FUNCTION_BLOCK _ETcVnBarcodeSearchDirection_TestSuite EXTENDS TcUnit.FB_TestSuite
VAR
END_VAR

TestAddress();
TestClearReference();
TestClone();
TestTypeNameReturnsExpected();
TestIdentifierReturnsExpected();
TestMakeReferenceToFollowsReference();
TestMakeReferenceToUpdatesReference();
TestSize();
TestValueReturnsExpectedAfterInit();
TestValueReturnsExpectedAfterChange();
TestSerializeTypeWith();
TestSerializeWith();
TestTryDeserializeFrom();
TestTryMakeReferenceToFollowsReference();
TestTryMakeReferenceToUpdatesReference();

METHOD PUBLIC TestAddress
VAR
    _type : _ETcVnBarcodeSearchDirection(ETcVnBarcodeSearchDirection.TCVN_BSD_ANY);
    notExpected : PVOID := 0;
    actual : PVOID;
END_VAR
TEST('TestAddress');

actual := _type.Address;

AssertFalse(
    Condition := (notExpected = actual),
    Message := 'Type did not return a valid address.'
);

TEST_FINISHED();
END_METHOD

METHOD PUBLIC TestClearReference
VAR
    _type : _ETcVnBarcodeSearchDirection(ETcVnBarcodeSearchDirection.TCVN_BSD_ANY);
	target : ETcVnBarcodeSearchDirection := ETcVnBarcodeSearchDirection.TCVN_BSD_ANY;
    expected : ETcVnBarcodeSearchDirection := ETcVnBarcodeSearchDirection.TCVN_BSD_ANY;
    actual : ETcVnBarcodeSearchDirection;
END_VAR
TEST('TestClearReference');

_type.MakeReferenceTo(target);
_type.ClearReference();
target := ETcVnBarcodeSearchDirection.TCVN_BSD_HORIZONTAL;

actual := _type.Value;

AssertEquals(
    Expected := expected,
    Actual := actual,
    Message := 'Value continued to follow target.'
);

TEST_FINISHED();
END_METHOD

METHOD PUBLIC TestClone
VAR
    _type : _ETcVnBarcodeSearchDirection(ETcVnBarcodeSearchDirection.TCVN_BSD_ANY);
	clone : I_Datatype;
	isValidClone : BOOL;
	compareResult : DINT;
END_VAR
TEST('TestClone');

clone := _type.Clone();

isValidClone := clone <> 0;

IF isValidClone THEN
	compareResult := memcmp(_type.Address, clone.Address, clone.Size);
END_IF

AssertTrue(
	Condition := isValidClone,
	Message := 'Clone did not produce a clone'
);

AssertEquals_DINT(
	Expected := 0,
    Actual := compareResult,
    Message := 'Clone did not return a valid clone.'
);

clone.Dispose();

TEST_FINISHED();
END_METHOD

METHOD PUBLIC TestIdentifierReturnsExpected
VAR
    _type : _ETcVnBarcodeSearchDirection(ETcVnBarcodeSearchDirection.TCVN_BSD_ANY);
    expected : STRING := 'ETcVnBarcodeSearchDirection';
    actual : STRING;
END_VAR
TEST('TestIdentifierReturnsExpected');

actual := _type.Identifier;

AssertEquals_STRING(
    Expected := expected,
    Actual := actual,
    Message := 'Type did not return correct iec type.'
);

TEST_FINISHED();
END_METHOD

METHOD PUBLIC TestMakeReferenceToFollowsReference
VAR
    _type : _ETcVnBarcodeSearchDirection(ETcVnBarcodeSearchDirection.TCVN_BSD_ANY);
	target : ETcVnBarcodeSearchDirection := ETcVnBarcodeSearchDirection.TCVN_BSD_ANY;
    expected : ETcVnBarcodeSearchDirection := ETcVnBarcodeSearchDirection.TCVN_BSD_HORIZONTAL;
    actual : ETcVnBarcodeSearchDirection;
END_VAR
TEST('TestMakeReferenceToFollowsReference');

_type.MakeReferenceTo(target);
target := ETcVnBarcodeSearchDirection.TCVN_BSD_HORIZONTAL;

actual := _type.Value;

AssertEquals(
    Expected := expected,
    Actual := actual,
    Message := 'Value did not follow target change.'
);

TEST_FINISHED();
END_METHOD

METHOD PUBLIC TestMakeReferenceToUpdatesReference
VAR
    _type : _ETcVnBarcodeSearchDirection(ETcVnBarcodeSearchDirection.TCVN_BSD_ANY);
	target : ETcVnBarcodeSearchDirection := ETcVnBarcodeSearchDirection.TCVN_BSD_ANY;
    expected : ETcVnBarcodeSearchDirection := ETcVnBarcodeSearchDirection.TCVN_BSD_HORIZONTAL;
    actual : ETcVnBarcodeSearchDirection;
END_VAR
TEST('TestMakeReferenceToUpdatesReference');

_type.MakeReferenceTo(target);
_type.Value := ETcVnBarcodeSearchDirection.TCVN_BSD_HORIZONTAL;

actual := target;

AssertEquals(
    Expected := expected,
    Actual := actual,
    Message := 'Value did not update target.'
);

TEST_FINISHED();
END_METHOD

METHOD PUBLIC TestSerializeTypeWith
VAR
    _type : _ETcVnBarcodeSearchDirection(ETcVnBarcodeSearchDirection.TCVN_BSD_ANY);
    serializer : JsonSerializer;
    expected : STRING(500) := '{"typeName":"ENUM","identifier":"ETcVnBarcodeSearchDirection","enumerations":["TCVN_BSD_ANY","TCVN_BSD_HORIZONTAL","TCVN_BSD_VERTICAL"],"baseType":{"typeName":"UDINT","minValue":0,"maxValue":4294967295,"isSigned":false,"isFloat":false}}'; 
    actual : STRING(500);
END_VAR
TEST('TestSerializeTypeWith');

serializer.Reset();
_type.SerializeTypeWith(serializer);
serializer.TryGetSerializedData(ADR(actual), SIZEOF(actual));

AssertEquals_STRING(
    Expected := expected,
    Actual := actual,
    Message := 'Serialization of type did not return correct string.'
);

TEST_FINISHED();
END_METHOD

METHOD PUBLIC TestSerializeWith
VAR
    _type : _ETcVnBarcodeSearchDirection(ETcVnBarcodeSearchDirection.TCVN_BSD_ANY);
    serializer : JsonSerializer;
    expected : STRING := '"TCVN_BSD_ANY"';
    actual : STRING(500);
END_VAR
TEST('TestSerializeWith');

serializer.Reset();
_type.SerializeWith(serializer);
serializer.TryGetSerializedData(ADR(actual), SIZEOF(actual));

AssertEquals_STRING(
    Expected := expected,
    Actual := actual,
    Message := 'Serialization of type data did not return correct string.'
);

TEST_FINISHED();
END_METHOD

METHOD PUBLIC TestSize
VAR
    _type : _ETcVnBarcodeSearchDirection(ETcVnBarcodeSearchDirection.TCVN_BSD_ANY);
    expected : UDINT := SIZEOF(ETcVnBarcodeSearchDirection);
    actual : UDINT;
END_VAR
TEST('TestSize');

actual := _type.Size;

AssertEquals_UDINT(
    Expected := Expected,
    Actual := actual,
    Message := 'Type did not return the correct size.'
);

TEST_FINISHED();
END_METHOD

METHOD PUBLIC TestTryDeserializeFrom
VAR
    deserializer : JsonDeserializer;
    feedback : DeserializerFeedback;
    json : STRING := '"TCVN_BSD_ANY"';
    _type : _ETcVnBarcodeSearchDirection(ETcVnBarcodeSearchDirection.TCVN_BSD_ANY);
    expected : ETcVnBarcodeSearchDirection := ETcVnBarcodeSearchDirection.TCVN_BSD_ANY;
    actual : ETcVnBarcodeSearchDirection;
 END_VAR
TEST('TestTryDeserializeFrom');

deserializer.Reset();
deserializer.TryLoad(json);
_type.TryDeserializeFrom(Deserializer, Feedback);

actual := _type.Value;

AssertEquals(
    Expected := expected,
    Actual := actual,
    Message := 'Type did not deserialize correctly.'
);

TEST_FINISHED();
END_METHOD

METHOD PUBLIC TestTryMakeReferenceToFollowsReference
VAR
    _type : _ETcVnBarcodeSearchDirection(ETcVnBarcodeSearchDirection.TCVN_BSD_ANY);
	target : _ETcVnBarcodeSearchDirection(ETcVnBarcodeSearchDirection.TCVN_BSD_ANY);
    expected : ETcVnBarcodeSearchDirection := ETcVnBarcodeSearchDirection.TCVN_BSD_HORIZONTAL;
    actual : ETcVnBarcodeSearchDirection;
END_VAR
TEST('TestTryMakeReferenceToFollowsReference');

_type.TryMakeReferenceTo(target);
target.Value := ETcVnBarcodeSearchDirection.TCVN_BSD_HORIZONTAL;

actual := _type.Value;

AssertEquals(
    Expected := expected,
    Actual := actual,
    Message := 'Value did not follow target change.'
);

TEST_FINISHED();
END_METHOD

METHOD PUBLIC TestTryMakeReferenceToUpdatesReference
VAR
    _type : _ETcVnBarcodeSearchDirection(ETcVnBarcodeSearchDirection.TCVN_BSD_ANY);
	target : _ETcVnBarcodeSearchDirection(ETcVnBarcodeSearchDirection.TCVN_BSD_ANY);
    expected : ETcVnBarcodeSearchDirection := ETcVnBarcodeSearchDirection.TCVN_BSD_HORIZONTAL;
    actual : ETcVnBarcodeSearchDirection;
END_VAR
TEST('TestTryMakeReferenceToUpdatesReference');

_type.TryMakeReferenceTo(target);
_type.Value := ETcVnBarcodeSearchDirection.TCVN_BSD_HORIZONTAL;

actual := target.Value;

AssertEquals(
    Expected := expected,
    Actual := actual,
    Message := 'Value did not update target.'
);

TEST_FINISHED();
END_METHOD

METHOD PUBLIC TestTypeNameReturnsExpected
VAR
    _type : _ETcVnBarcodeSearchDirection(ETcVnBarcodeSearchDirection.TCVN_BSD_ANY);
    expected : STRING := 'ENUM';
    actual : STRING;
END_VAR
TEST('TestTypeNameReturnsExpected');

actual := _type.TypeName;

AssertEquals_STRING(
    Expected := expected,
    Actual := actual,
    Message := 'Type did not return correct iec type.'
);

TEST_FINISHED();
END_METHOD

METHOD PUBLIC TestValueReturnsExpectedAfterChange
VAR
    _type : _ETcVnBarcodeSearchDirection(ETcVnBarcodeSearchDirection.TCVN_BSD_ANY);
    expected : ETcVnBarcodeSearchDirection := ETcVnBarcodeSearchDirection.TCVN_BSD_HORIZONTAL;
    actual : ETcVnBarcodeSearchDirection;
END_VAR
TEST('TestValueReturnsExpectedAfterChange');

_type.Value := ETcVnBarcodeSearchDirection.TCVN_BSD_HORIZONTAL;

actual := _type.Value;

AssertEquals(
    Expected := expected,
    Actual := actual,
    Message := 'Expected value not returned after change.'
);

TEST_FINISHED();
END_METHOD

METHOD PUBLIC TestValueReturnsExpectedAfterInit
VAR
    _type : _ETcVnBarcodeSearchDirection(ETcVnBarcodeSearchDirection.TCVN_BSD_ANY);
    expected : ETcVnBarcodeSearchDirection := ETcVnBarcodeSearchDirection.TCVN_BSD_ANY;
    actual : ETcVnBarcodeSearchDirection;
END_VAR
TEST('TestValueReturnsExpectedAfterInit');

actual := _type.Value;

AssertEquals(
    Expected := expected,
    Actual := actual,
    Message := 'Expected value not returned after Init.'
);

TEST_FINISHED();
END_METHOD

END_FUNCTION_BLOCK

(* stored: Version 1.1.0.1, ProductVersion 3.1.4024.12
   POU _ETcVnBarcodeSearchDirection_TestSuite: Id {e74ac28e-284a-055c-2f79-e519c7e46c32}, SpecialFunc None
   Method TestAddress: Id {2e7cf123-4be8-0228-21c3-6144339cca67}
   Method TestClearReference: Id {5fe629c4-5d82-0fba-14be-2622c73a5dea}
   Method TestClone: Id {e27b567b-0e02-0726-3f47-982c269e6a9f}
   Method TestIdentifierReturnsExpected: Id {2f8a9b83-4eff-037c-1235-9039576edc79}
   Method TestMakeReferenceToFollowsReference: Id {72aa7b61-c70e-0e07-34ad-2961b41ab574}
   Method TestMakeReferenceToUpdatesReference: Id {578f5f45-390f-017f-05b9-0e060e9d77ed}
   Method TestSerializeTypeWith: Id {f37fd8ed-a2d1-09b4-396d-2e7983bb9016}
   Method TestSerializeWith: Id {f1f1af51-12b0-0fe5-0734-fbafab1a0651}
   Method TestSize: Id {6be10135-8162-09ac-2b2c-389585891502}
   Method TestTryDeserializeFrom: Id {b63ddfa5-1487-0d34-07f2-1ded02acfd35}
   Method TestTryMakeReferenceToFollowsReference: Id {cef35bfd-b866-0475-28bd-4e8270ae56a7}
   Method TestTryMakeReferenceToUpdatesReference: Id {f9547cc7-c4e5-0139-0973-7970019f21d0}
   Method TestTypeNameReturnsExpected: Id {add9fa52-eb0d-0791-059b-089a372652c6}
   Method TestValueReturnsExpectedAfterChange: Id {9d79bc52-a79c-0e8c-14ac-b8f36c767f58}
   Method TestValueReturnsExpectedAfterInit: Id {4bc13dae-2f58-0740-2e66-6d372eef73a0} *)
